{region '#Template'}
	{attribute 'Version' := '1.0.0.0'}
	{attribute 'Tags' := '"LCID": "1031", "Text": "Trade, Plant, Heating System"'}
	{attribute 'Tags' := '"LCID": "1033", "Text": "Trade, Plant, Heating System"'}
	{attribute 'Description' := '"LCID": "1031", "Text": "Aufruf der Anlagen des Gewerks Heizsysteme"'}
	{attribute 'Description' := '"LCID": "1033", "Text": "Calling the plants of the trade heating system"'}
{endregion}
FUNCTION_BLOCK FB_BA_H EXTENDS FB_BA_View
VAR_INPUT CONSTANT
	HTC01				: FB_BA_H_HtgCir01;		
END_VAR
VAR_INPUT
END_VAR
VAR_OUTPUT
END_VAR
VAR
END_VAR

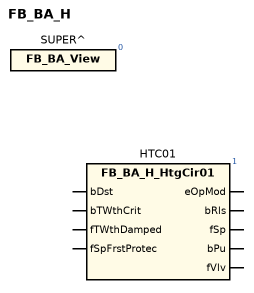
SUPER^(); // FB_BA_View
HTC01(); // FB_BA_H_HtgCir01

METHOD FB_init : BOOL
VAR_INPUT
	bInitRetains : BOOL; // if TRUE, the retain variables are initialized (warm start / cold start)
	bInCopyCode : BOOL;  // if TRUE, the instance afterwards gets moved into the copy code (online change)
END_VAR
HTC01.iParent 					:= THIS^;	
HTC01.sObjectName				:= CONCAT(TxTPlant_Heating_circuit_sObjectName,'01');							
HTC01.sDescription				:= TxTPlant_Heating_circuit_sDescription;	
HTC01.eDPADMode					:= E_BA_DPADMode.eInclude;

HTC01.GeneralSettings.Subject	:= Site.GeneralSettings_Subject;
HTC01.GeneralSettings.sTarget	:= Site.GeneralSettings_NetId;
END_METHOD

END_FUNCTION_BLOCK

(* stored: Version 1.1.0.1, ProductVersion 3.1.4024.9
   POU FB_BA_H: Id {8d62bf85-3048-4c48-af2b-62938abe3d12}, SpecialFunc None
   Method FB_init: Id {83e05d5a-fbe8-4426-b007-bab3b83c45ac} *)
